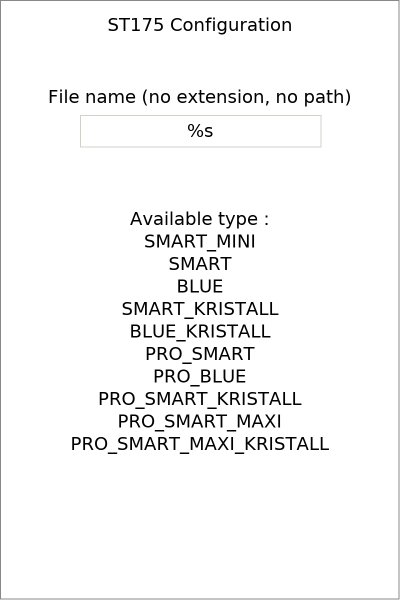
VISUALIZATION VISU_Recipe_ST175  // 400x600
    Textfield (80,115 241x32), "%s", text variable: _20_AUTO.recipe.st175.file_name
        OnMouseDown: write the text variable via Default
    Label (0,5 400x40), "ST175 Configuration"
    Label (24,87 352x20), "File name (no extension, no path)"
    Label (59,177 282x309), "Available type : SMART_MINI SMART BLUE SMART_KRISTALL BLUE_KRISTALL PRO_SMART PRO_BLUE PRO_SMART_KRISTALL PRO_SMART_MAXI PRO_SMART_MAXI_KRISTALL"
END_VISUALIZATION

(* stored: Version 1.1.0.1, ProductVersion 3.1.4024.6
   Visu VISU_Recipe_ST175: Id {9bcd3d30-c5e5-480c-a76b-bccd1c299c77} *)
